(* PLC project SafeLOGIC, BrAutomation SafeDESIGNER  5.24.1.0 *)
(* stored: companyURL http://www.br-automation.com, creationDateTime Fri Nov 28 15:07:09 2025 *)

PROGRAM PLAUSIBILITY
  VAR  (* added by the conversion: wires and edge detectors of the diagram *)
    _OR_S4_OUT : BOOL;
    _SAFEBOOL_TO_BOOL17_OUT : BOOL;
  END_VAR

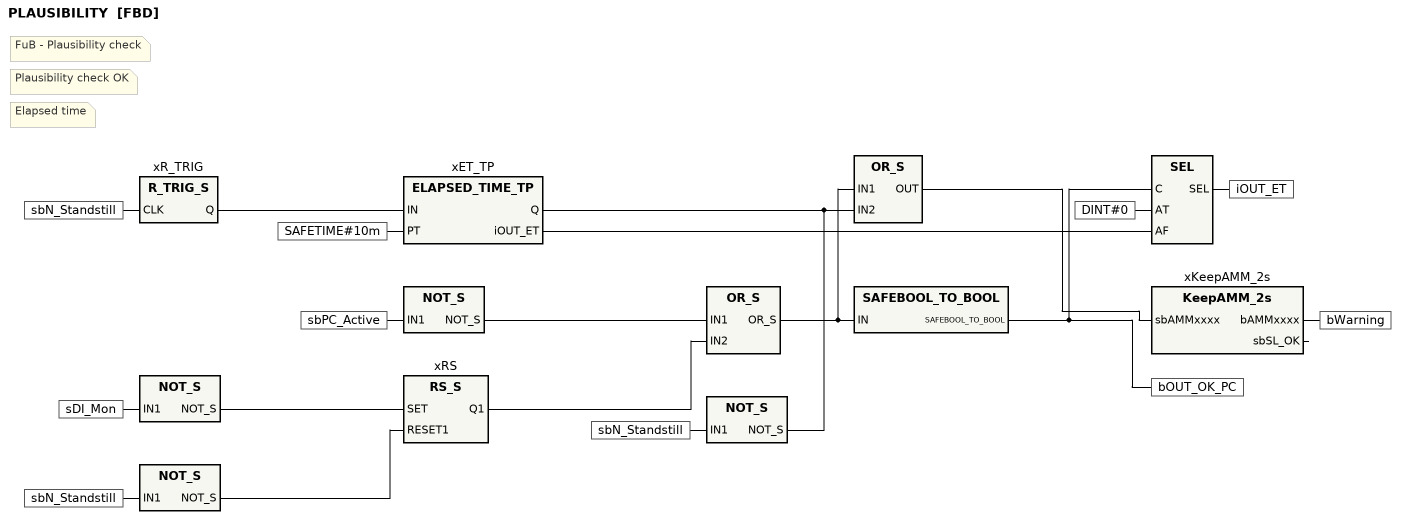
(* FBD diagram, written out as Structured Text *)
(* FuB - Plausibility check *)
(* Plausibility check OK *)
xRS(SET := NOT_S(sDI_Mon), RESET1 := NOT_S(sbN_Standstill));
_OR_S4_OUT := OR_S(NOT_S(sbPC_Active), xRS.Q1);
_SAFEBOOL_TO_BOOL17_OUT := SAFEBOOL_TO_BOOL(_OR_S4_OUT);
bOUT_OK_PC := _SAFEBOOL_TO_BOOL17_OUT;
xR_TRIG(CLK := sbN_Standstill);
xET_TP(IN := xR_TRIG.Q, PT := SAFETIME#10m);
xKeepAMM_2s(sbAMMxxxx := OR_S(_OR_S4_OUT, NOT_S(sbN_Standstill), xET_TP.Q));
bWarning := xKeepAMM_2s.bAMMxxxx;
(* Elapsed time *)
iOUT_ET := SEL(_SAFEBOOL_TO_BOOL17_OUT, DINT#0, xET_TP.iOUT_ET);
END_PROGRAM
